(* IEC 61131-3 sources: com.logicals.lc3.webinar/usRTS_RPMControl_iSOC/src_FB_LIB_SAFE/Convert/INT, 4 files *)

(* ---- wINT_TO_DINT.iecst ---- *)
NAMESPACE logicals.web.standard
NAMESPACE convert

/*
 * Function block wrapper for IEC 61131-3 TO_DINT<br>
 * IN =  input value (INT)<br>
 * OUT = IN (DINT)<br>
 */
FUNCTION_BLOCK wINT_TO_DINT
	{ vNameAlignment:="center"; altName:="INT_TO_DINT"; bgColor:="LightPink"; width:=140; hideIONames; }
	VAR_INPUT
		IN : INT;
	END_VAR
	VAR_OUTPUT
		OUT: DINT;
	END_VAR

	OUT := TO_DINT(IN:=IN, ENO=>ENO);
END_FUNCTION_BLOCK

END_NAMESPACE
END_NAMESPACE

(* ---- wINT_TO_LINT.iecst ---- *)
NAMESPACE logicals.web.standard
NAMESPACE convert

/*
 * Function block wrapper for IEC 61131-3 TO_LINT<br>
 * IN =  input value (INT)<br>
 * OUT = IN (LINT)<br>
 */
FUNCTION_BLOCK wINT_TO_LINT
	{ vNameAlignment:="center"; altName:="INT_TO_LINT"; bgColor:="LightPink"; width:=140; hideIONames; }
	VAR_INPUT
		IN : INT;
	END_VAR
	VAR_OUTPUT
		OUT: LINT;
	END_VAR

	OUT := TO_LINT(IN:=IN, ENO=>ENO);
END_FUNCTION_BLOCK

END_NAMESPACE
END_NAMESPACE

(* ---- wTRUNC_INT_TO_SINT.iecst ---- *)
NAMESPACE logicals.web.standard
NAMESPACE convert

/*
 * Function block wrapper for IEC 61131-3 TO_SINT<br>
 * IN =  input value (INT)<br>
 * OUT = IN (SINT)<br>
 */
FUNCTION_BLOCK wTRUNC_INT_TO_SINT
	{ vNameAlignment:="center"; altName:="TRUNC_INT_TO_SINT"; bgColor:="LightPink"; width:=180; hideIONames; }
	VAR_INPUT
		IN : INT;
	END_VAR
	VAR_OUTPUT
		OUT: SINT;
	END_VAR

	OUT := TO_SINT(IN:=IN, ENO=>ENO);
END_FUNCTION_BLOCK

END_NAMESPACE
END_NAMESPACE

(* ---- wTRUNC_INT_TO_UINT.iecst ---- *)
NAMESPACE logicals.web.standard
NAMESPACE convert

/*
 * Function block wrapper for IEC 61131-3 TO_UINT<br>
 * IN =  input value (INT)<br>
 * OUT = IN (UINT)<br>
 */
FUNCTION_BLOCK wTRUNC_INT_TO_UINT
	{ vNameAlignment:="center"; altName:="TRUNC_INT_TO_UINT"; bgColor:="Plum"; width:=180; hideIONames; }
	VAR_INPUT
		IN : INT;
	END_VAR
	VAR_OUTPUT
		OUT: UINT;
	END_VAR

	OUT := TO_UINT(IN:=IN, ENO=>ENO);
END_FUNCTION_BLOCK

END_NAMESPACE
END_NAMESPACE
